FUNCTION_BLOCK FB_Convert_2WindDir
VAR_INPUT
	iInput			:	INT;
	tRefresh		:	TIME;
END_VAR
VAR_OUTPUT
	wOut			:	WORD;
END_VAR
VAR
	rX				:	REAL;
	tonBlock		:	TON;
END_VAR


tonBlock(IN := NOT tonBlock.Q, PT := tRefresh);

IF tonBlock.Q THEN

	rX := iInput / 91.019; //Annahme 360° entspr. 32767
	wOut := REAL_TO_WORD(rX);
	
END_IF

END_FUNCTION_BLOCK

(* stored: Version 1.1.0.1, ProductVersion 3.1.4024.13
   POU FB_Convert_2WindDir: Id {720830b7-668f-4ba3-b9f5-d41ab53d764c}, SpecialFunc None *)
